FUNCTION_BLOCK GoodFeaturesToTrack (* openCV goodFeaturesToTrack *)
  (* Version 1.0, AN, SWDC RTSoft *)
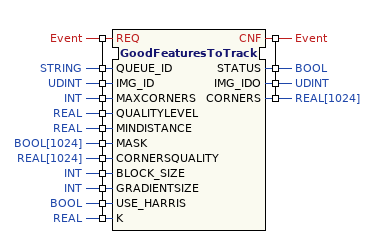
  EVENT_INPUT
    REQ WITH QUEUE_ID, IMG_ID, MAXCORNERS, QUALITYLEVEL, MINDISTANCE, MASK, CORNERSQUALITY, BLOCK_SIZE, GRADIENTSIZE, USE_HARRIS, K;
  END_EVENT
  EVENT_OUTPUT
    CNF WITH STATUS, IMG_IDO, CORNERS;
  END_EVENT
  VAR_INPUT
    QUEUE_ID : STRING;
    IMG_ID : UDINT;
    MAXCORNERS : INT;
    QUALITYLEVEL : REAL;
    MINDISTANCE : REAL;
    MASK : ARRAY [0..1023] OF BOOL;
    CORNERSQUALITY : ARRAY [0..1023] OF REAL;
    BLOCK_SIZE : INT;
    GRADIENTSIZE : INT;
    USE_HARRIS : BOOL;
    K : REAL;
  END_VAR
  VAR_OUTPUT
    STATUS : BOOL;
    IMG_IDO : UDINT;
    CORNERS : ARRAY [0..1023] OF REAL;
  END_VAR
  ALGORITHM REQ IN ST:

  END_ALGORITHM
END_FUNCTION_BLOCK
